(* Schneider Machine Expert - Basic project City_Zone, file version 1.8.0.0 *)
(* ProjectInformations: Name=New project *)

HARDWARE
  Cpu 0: TM221CE16R
  EthernetConfiguration: NetworkName=M221, IpAllocationMode=FixedAddress, IpAddress=172.18.212.88, SubnetMask=255.255.255.0
  SerialLineConfiguration: Baud=Baud19200, Parity=ParityEven, DataBits=DataBits8, StopBits=StopBits1, PhysicalMedium=PhysicalMediumRs485, TransmissionMode=TransmissionModeModbusRtu, SlaveId=1, Addressing=SlaveAddressing
  MastTask: UsePeriodScanMode=false, PeriodScan=100
  FastTask: Period=255
  CpuBehavior: StartingMode=StartAsPreviousState, AutoSaveRamOnEeprom=true, WatchdogPeriod=250

SYMBOLS  (address, symbol, comment, settings)
  %M30        "Choose Attack Scenario"
  %Q0.0       "Tournout Control A"
  %Q0.1       "Track A"
  %Q0.2       "Track B"
  %Q0.3       "Track B"
  %Q0.4       "Track B"
  %Q0.5       "Red Light"
  %Q0.6       "White Light"

POU New POU
  (* SectionNumber=1 *)

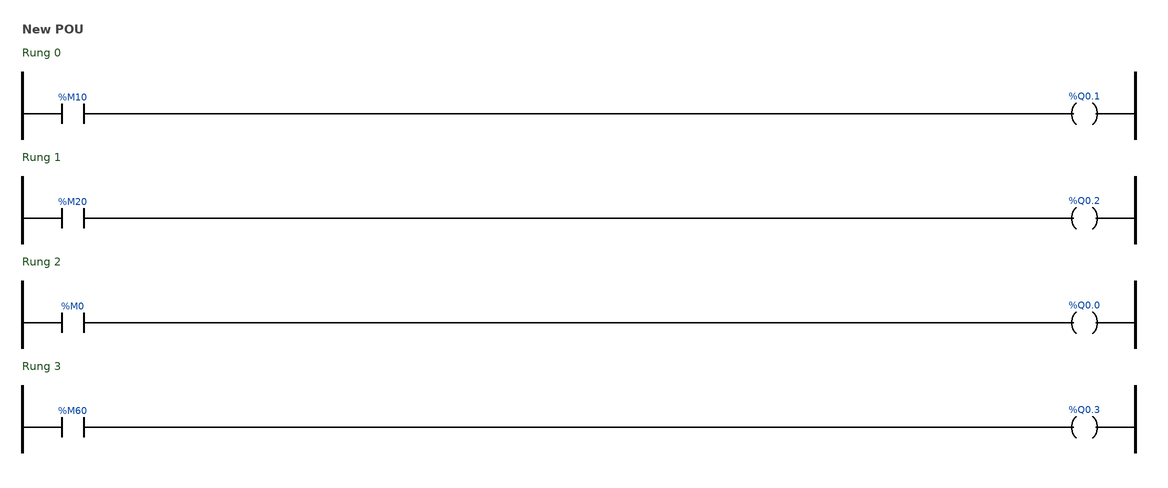

// Rung 0
  LD %M10
  ST %Q0.1
  // as ST:
  //   %Q0.1 := %M10;

// Rung 1
  LD %M20
  ST %Q0.2
  // as ST:
  //   %Q0.2 := %M20;

// Rung 2
  LD %M0
  ST %Q0.0
  // as ST:
  //   %Q0.0 := %M0;

// Rung 3
  LD %M60
  ST %Q0.3
  // as ST:
  //   %Q0.3 := %M60;
